// TIA Portal V17 export
// export: Created 2023-04-03T06:31:31.3801066Z, ExportSetting WithDefaults, DisplayName Totally Integrated Automation Portal, DisplayVersion V17 Update 4, DisplayName TIA Portal Openness, DisplayVersion V17 Update 4, DisplayName TIA Portal Version Control Interface, DisplayVersion V17, DisplayName STEP 7 Professional, DisplayVersion V17 Update 4, DisplayName STEP 7 Safety, DisplayVersion V17, DisplayName WinCC Professional, DisplayVersion V17 Update 4
FUNCTION "EthernetDiag" : Void   // FC401, LAD
TITLE = Ethernet Diagnostic
{ S7_Optimized_Access := 'TRUE' }
VERSION : 0.1
// stored: AutoNumber false, IsIECCheckEnabled false, SetENOAutomatically false, UDAEnableTagReadback false
BEGIN

REGION Network 1: Ethernet Diagnostic PLC PEMS
   // Block to check ethernet connection to PEMS (used in HMI)
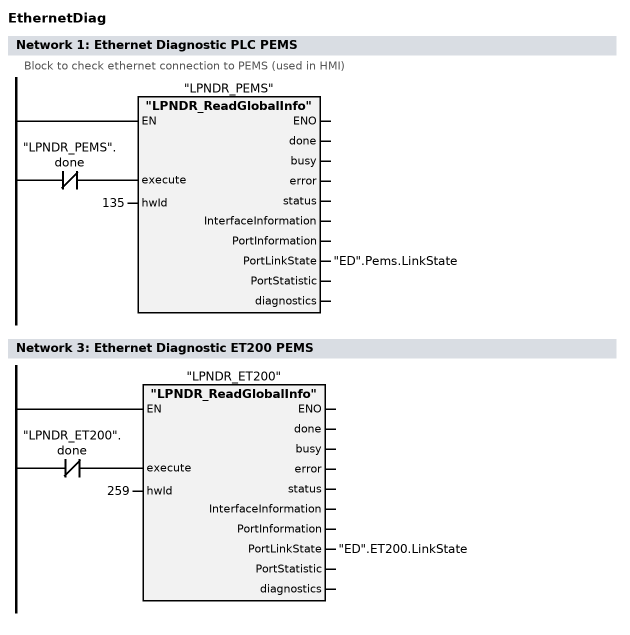
   RUNG wire#powerrail
      "LPNDR_PEMS"(execute := wire#w1, hwId := 135, done =>, busy =>, error =>, status =>, InterfaceInformation =>, PortInformation =>, PortLinkState => "ED".Pems.LinkState, PortStatistic =>, diagnostics =>)
   END_RUNG
   RUNG wire#powerrail
      I_Contact( "LPNDR_PEMS".done )
   END_RUNG wire#w1
   // the same network as SCL:
   "LPNDR_PEMS"(execute := NOT "LPNDR_PEMS".done, hwId := 135, PortLinkState => "ED".Pems.LinkState);   // "LPNDR_ReadGlobalInfo"
END_REGION

REGION Network 2 (SCL): Ethernet Diagnostic PLC PEMS
   "ED".Pems.X1 := "ED".Pems.LinkState[1].portLinkState = 1;
   "ED".Pems.X2 := "ED".Pems.LinkState[2].portLinkState = 1;
   "ED".Pems.X3 := "ED".Pems.LinkState[3].portLinkState = 1;
END_REGION

REGION Network 3: Ethernet Diagnostic ET200 PEMS
   RUNG wire#powerrail
      "LPNDR_ET200"(execute := wire#w1, hwId := 259, done =>, busy =>, error =>, status =>, InterfaceInformation =>, PortInformation =>, PortLinkState => "ED".ET200.LinkState, PortStatistic =>, diagnostics =>)
   END_RUNG
   RUNG wire#powerrail
      I_Contact( "LPNDR_ET200".done )
   END_RUNG wire#w1
   // the same network as SCL:
   "LPNDR_ET200"(execute := NOT "LPNDR_ET200".done, hwId := 259, PortLinkState => "ED".ET200.LinkState);   // "LPNDR_ReadGlobalInfo"
END_REGION

REGION Network 4 (SCL): Ethernet Diagnostic ET200 PEMS
   "ED".ET200.X1 := "ED".ET200.LinkState[1].portLinkState = 1;
   "ED".ET200.X2 := "ED".ET200.LinkState[2].portLinkState = 1;
END_REGION
END_FUNCTION
